{attribute 'linkalways'} 
{attribute 'no_explicit_call' := 'This FB is a CLASS and must be accessed using methods or properties'}
{attribute 'enable_dynamic_creation'}
FUNCTION_BLOCK FINAL NE_UDINT EXTENDS Node
VAR
	in1 : _UDINT(0);
	in2 : _UDINT(0);
	out : _BOOL(FALSE);
END_VAR

METHOD PUBLIC Clone : I_Node
VAR
	pNode : POINTER TO NE_UDINT;
END_VAR
pNode := __NEW(NE_UDINT);
Clone := pNode^;
END_METHOD

METHOD FB_init : BOOL
VAR_INPUT
	bInitRetains : BOOL; // if TRUE, the retain variables are initialized (warm start / cold start)
	bInCopyCode : BOOL;  // if TRUE, the instance afterwards gets moved into the copy code (online change)
END_VAR
AddInput('in1',THIS^.in1);
AddInput('in2',THIS^.in2);
AddOutput('out', THIS^.out);
END_METHOD

METHOD PROTECTED OnExecute
VAR
END_VAR
out.Value := in1.Value <> in2.Value;
END_METHOD

END_FUNCTION_BLOCK

(* stored: Version 1.1.0.1, ProductVersion 3.1.4024.15
   POU NE_UDINT: Id {af08bbe4-3317-4211-8120-f67e4ccf2673}, SpecialFunc None
   Folder Constructor: Id {4950f6a6-297e-4654-936b-235a453351af}
   Method Clone: Id {05125dfa-21fc-45de-868d-f48ea3bdce24}
   Method FB_init: Id {c3778c61-8298-447f-b872-20f436a469f5}
   Method OnExecute: Id {9ed91b56-4690-4863-8e75-667c13da6ea9} *)
